// TIA Portal V18 export
FUNCTION "OutputMapping" : Void   // FC14, LAD
{ S7_Optimized_Access := 'TRUE' }
VERSION : 0.1
// stored: AutoNumber true, IsIECCheckEnabled false, SetENOAutomatically false, UDAEnableTagReadback false
   VAR_TEMP
      tempNotConnect : Bool;
   END_VAR
BEGIN

REGION Network 1: Output CC - Betriebsart
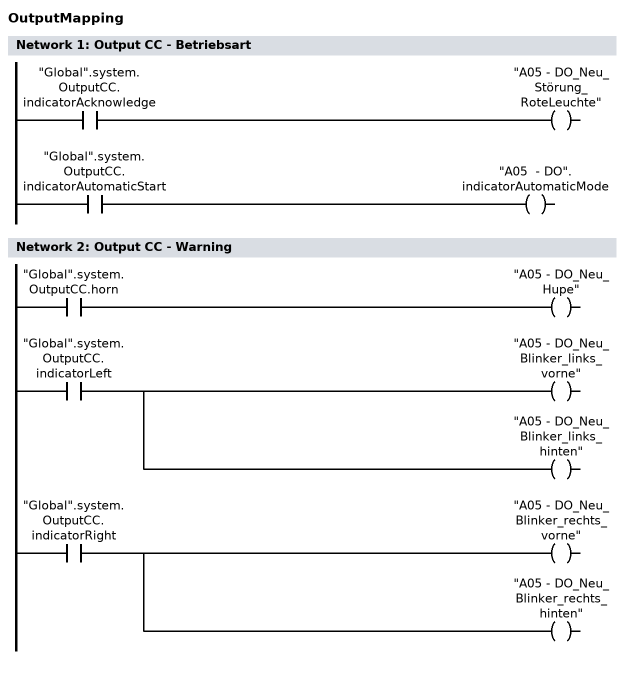
   RUNG wire#powerrail
      Contact( "Global".system.OutputCC.indicatorAcknowledge )
      Coil( "A05 - DO_Neu_Störung_RoteLeuchte" )
   END_RUNG
   RUNG wire#powerrail
      Contact( "Global".system.OutputCC.indicatorAutomaticStart )
      Coil( "A05  - DO".indicatorAutomaticMode )
   END_RUNG
   // the same network as SCL:
   "A05 - DO_Neu_Störung_RoteLeuchte" := "Global".system.OutputCC.indicatorAcknowledge;
   "A05  - DO".indicatorAutomaticMode := "Global".system.OutputCC.indicatorAutomaticStart;
END_REGION

REGION Network 2: Output CC - Warning
   RUNG wire#powerrail
      Contact( "Global".system.OutputCC.horn )
      Coil( "A05 - DO_Neu_Hupe" )
   END_RUNG
   RUNG wire#powerrail
      Contact( "Global".system.OutputCC.indicatorLeft )
      wire#w1
      Coil( "A05 - DO_Neu_Blinker_links_vorne" )
   END_RUNG
   RUNG wire#w1
      Coil( "A05 - DO_Neu_Blinker_links_hinten" )
   END_RUNG
   RUNG wire#powerrail
      Contact( "Global".system.OutputCC.indicatorRight )
      wire#w2
      Coil( "A05 - DO_Neu_Blinker_rechts_vorne" )
   END_RUNG
   RUNG wire#w2
      Coil( "A05 - DO_Neu_Blinker_rechts_hinten" )
   END_RUNG
   // the same network as SCL:
   "A05 - DO_Neu_Hupe" := "Global".system.OutputCC.horn;
   "A05 - DO_Neu_Blinker_links_vorne" := "Global".system.OutputCC.indicatorLeft;
   "A05 - DO_Neu_Blinker_links_hinten" := "Global".system.OutputCC.indicatorLeft;
   "A05 - DO_Neu_Blinker_rechts_vorne" := "Global".system.OutputCC.indicatorRight;
   "A05 - DO_Neu_Blinker_rechts_hinten" := "Global".system.OutputCC.indicatorRight;
END_REGION
END_FUNCTION
